KUKA KRL program: Calibration_2.src

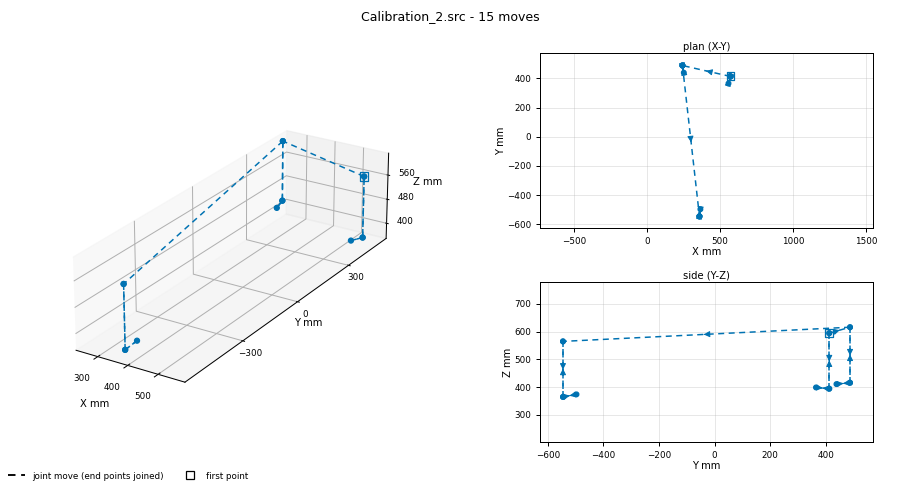
[picture p0: tool path of Calibration_2.src, 15 of 17 moves have a stored position in this frame; points joined in program order, loops and branches not executed]
&ACCESS RVP
&REL 1
&PARAM TEMPLATE = C:\KRC\Roboter\Template\vorgabe
&PARAM EDITMASK = *
DEF Calibration_2 ( )


;FOLD INI
;FOLD BASISTECH INI
GLOBAL INTERRUPT DECL 3 WHEN $STOPMESS==TRUE DO IR_STOPM ( )
INTERRUPT ON 3
BAS (#INITMOV,0 )
;ENDFOLD (BASISTECH INI)
;ENDFOLD (INI)

;FOLD STARTPOSITION - BASE IS 0, TOOL IS 5, SPEED IS 15%, POSITION IS A1 5,A2 -90,A3 100,A4 5,A5 -10,A6 -5,E1 0,E2 0,E3 0,E4 0
$BWDSTART = FALSE
PDAT_ACT = {VEL 15,ACC 100,APO_DIST 50}
FDAT_ACT = {TOOL_NO 5,BASE_NO 0,IPO_FRAME #BASE}
BAS (#PTP_PARAMS,15)
PTP  {A1 5,A2 -90,A3 100,A4 5,A5 -10,A6 -5,E1 0,E2 0,E3 0,E4 0}
;ENDFOLD

;FOLD LIN SPEED IS 0.1 m/sec, INTERPOLATION SETTINGS IN FOLD
$VEL.CP=0.1
$ADVANCE=3
;ENDFOLD

BAS(#VEL_PTP,10)
PTP {X 571.404, Y 413.048, Z 594.482, A -106.282, B -5.184, C -90.399, E1 0, E2 0, E3 0, E4 0, S 'B010'} C_PTP
PTP {X 571.404, Y 413.048, Z 394.482, A -106.282, B -5.184, C -90.399, E1 0, E2 0, E3 0, E4 0, S 'B010'} C_PTP
BAS(#VEL_PTP,2)
PTP {X 557.443, Y 365.25, Z 399, A -106.282, B -5.184, C -90.399, E1 0, E2 0, E3 0, E4 0, S 'B010'}
BAS(#VEL_PTP,10)
PTP {X 571.404, Y 413.048, Z 394.482, A -106.282, B -5.184, C -90.399, E1 0, E2 0, E3 0, E4 0, S 'B010'} C_PTP
PTP {X 571.404, Y 413.048, Z 594.482, A -106.282, B -5.184, C -90.399, E1 0, E2 0, E3 0, E4 0, S 'B010'} C_PTP
PTP {X 241.907, Y 487.887, Z 615.854, A -79.344, B 5.581, C -89.215, E1 0, E2 0, E3 0, E4 0, S 'B010'} C_PTP
PTP {X 241.907, Y 487.887, Z 415.854, A -79.344, B 5.581, C -89.215, E1 0, E2 0, E3 0, E4 0, S 'B010'} C_PTP
BAS(#VEL_PTP,2)
PTP {X 251.109, Y 438.982, Z 410.991, A -79.344, B 5.581, C -89.215, E1 0, E2 0, E3 0, E4 0, S 'B010'}
BAS(#VEL_PTP,10)
PTP {X 241.907, Y 487.887, Z 415.854, A -79.344, B 5.581, C -89.215, E1 0, E2 0, E3 0, E4 0, S 'B010'} C_PTP
PTP {X 241.907, Y 487.887, Z 615.854, A -79.344, B 5.581, C -89.215, E1 0, E2 0, E3 0, E4 0, S 'B010'} C_PTP
PTP {X 358.365, Y -545.782, Z 564.83, A 82.516, B -10.62, C -176.878, E1 0, E2 0, E3 0, E4 0, S 'B010'} C_PTP
PTP {X 358.365, Y -545.782, Z 364.83, A 82.516, B -10.62, C -176.878, E1 0, E2 0, E3 0, E4 0, S 'B010'} C_PTP
BAS(#VEL_PTP,2)
PTP {X 364.766, Y -497.057, Z 374.045, A 82.516, B -10.62, C -176.878, E1 0, E2 0, E3 0, E4 0, S 'B010'}
BAS(#VEL_PTP,10)
PTP {X 358.365, Y -545.782, Z 364.83, A 82.516, B -10.62, C -176.878, E1 0, E2 0, E3 0, E4 0, S 'B010'} C_PTP
PTP {X 358.365, Y -545.782, Z 564.83, A 82.516, B -10.62, C -176.878, E1 0, E2 0, E3 0, E4 0, S 'B010'} C_PTP
PTP {A1 5, A2 -90, A3 100, A4 5, A5 -10, A6 -5, E1 0, E2 0, E3 0, E4 0} C_PTP

END
